INTERFACE I_SourceLockable

METHOD LockSource : E_RpcMethodResponse
VAR_INPUT
    bLock : BOOL;
END_VAR
END_METHOD

END_INTERFACE

(* stored: Version 1.1.0.1, ProductVersion 3.1.4026.12
   Itf I_SourceLockable: Id {c0000003-0000-0000-0000-000000000001}
   Method LockSource: Id {c0000003-0000-0000-1000-000000000001} *)
